KUKA KRL data list: art_air.dat

&ACCESS RV2
DEFDAT  art_air PUBLIC
DECL INT low_air_signal_timer=0
DECL INT AIR_SIGNAL_OUT_TIME=2000
DECL GLOBAL BOOL ART_Air_low_preassure=FALSE
ENDDAT
